// TIA Portal V16 export
// export: Created 2022-04-09T12:33:16.9078898Z, ExportSetting WithDefaults, DisplayName Totally Integrated Automation Portal, DisplayVersion V16 Update 3, DisplayName TIA Portal Version Control Interface, DisplayVersion V16 Update 2, DisplayName TIA Portal Openness, DisplayVersion V16 Update 3, DisplayName STEP 7 Professional, DisplayVersion V16 Update 3, DisplayName STEP 7 Safety, DisplayVersion V16, DisplayName WinCC Professional, DisplayVersion V16 Update 3
TYPE "UT22001_Dy_InstAnalogRead"
TITLE = Dynamic UDT [INSTRUMENTATION] — Analog Instrument Read, Scale and Monitor
// PRACTICAL SERIES AUTOMATION LIBRARY (PAL)   —   COPYRIGHT 2020 – M. GLEDHILL (MIT LICENCE)
//                   ———— ◆ ————
// FULL ONLINE DOCUMENTATION IS AVAILABLE AT: https://practicalseries.com/2001-pal/index.html
// stored: IsFailsafeCompliant false
   STRUCT
      revInfo : "UT01000_St_SysRevision";   // Revision information
      ___________0010_0 { ExternalAccessible := 'False'; ExternalVisible := 'False'; ExternalWritable := 'False'} : Int;
      ___________0010_1 { ExternalAccessible := 'False'; ExternalVisible := 'False'; ExternalWritable := 'False'} : Int;   // ▀▀▀▀ STATUS (FOR BLOCK ICON AND SYMBOL)
      status_ConfigError : Bool;   // STATUS — Block is configured incorrectly
      status_Alm_H : Bool;   // STATUS — High alarm is active (1 = alarm active, 0 = no alarm)
      status_Alm_L : Bool;   // STATUS — Low alarm is active (1 = alarm active, 0 = no alarm)
      status_Wrn_H : Bool;   // STATUS — High warning is active (1 = warning active, 0 = no warning)
      status_Wrn_L : Bool;   // STATUS — Low warning is active (1 = warning active, 0 = no warning)
      status_Alm_H_Mask : Bool;   // STATUS — High alarm is masked (1 = alarm masked, 0 = normal)
      status_Alm_L_Mask : Bool;   // STATUS — Low alarm is masked (1 = alarm masked, 0 = normal)
      status_Wrn_H_Mask : Bool;   // STATUS — High warning is masked (1 = warning masked, 0 = normal)
      status_Wrn_L_Mask : Bool;   // STATUS — Low warning is masked (1 = warning masked, 0 = normal)
      status_Alm_H_Dis : Bool;   // STATUS — High alarm is disabled (1 = alarm disabled, 0 = normal)
      status_Alm_L_Dis : Bool;   // STATUS — Low alarm is disabled (1 = alarm disabled, 0 = normal)
      status_Wrn_H_Dis : Bool;   // STATUS — High warning is disabled (1 = warning disabled, 0 = normal)
      status_Wrn_L_Dis : Bool;   // STATUS — Low warning is disabled (1 = warning disabled, 0 = normal)
      status_Fault : Bool;   // STATUS — Device is in fault (1 = fault present, 0 = healthy)
      status_SimOn : Bool;   // STATUS — Device is in simulation mode (1 = simulation mode on, 0 = normal)
      status_RemoteOn : Bool;   // STATUS — Device is in remote mode (1 = remote mode, 0 = remote mode off)
      status_LocalOn : Bool;   // STATUS — Device is in local mode (1 = local mode, 0 = local mode off)
      status_RLOff : Bool;   // STATUS — Remote/local mode disabled (1 = ALL mode on, 0 = RL mode selected)
      ___________0020_0 { ExternalAccessible := 'False'; ExternalVisible := 'False'; ExternalWritable := 'False'} : Int;
      ___________0020_1 { ExternalAccessible := 'False'; ExternalVisible := 'False'; ExternalWritable := 'False'} : Int;   // ▀▀▀▀ CALCULATED VALUES (ABSOLUTE OVER AND UNDER RANGE)
      cal_OR_Abs : Real;   // CALC — Over-range limit (absolute value)
      cal_UR_Abs : Real;   // CALC — Under-range limit (absolute value)
      ___________0030_0 { ExternalAccessible := 'False'; ExternalVisible := 'False'; ExternalWritable := 'False'} : Int;
      ___________0030_2 { ExternalAccessible := 'False'; ExternalVisible := 'False'; ExternalWritable := 'False'} : Int;   // ▀▀▀▀ OPERATING MODE SELECTION (FROM FACEPLATE OR PANEL)
      mode_Alm_H_MaskOn : Bool;   // MODE — Mask Alm_H (1 = mask alarm, 0 = normal)
      mode_Alm_L_MaskOn : Bool;   // MODE — Mask Alm_L (1 = mask alarm, 0 = normal)
      mode_Wrn_H_MaskOn : Bool;   // MODE — Mask Wrn_H (1 = mask warning, 0 = normal)
      mode_Wrn_L_MaskOn : Bool;   // MODE — Mask Wrn_H (1 = mask warning, 0 = normal)
      mode_SimOn : Bool := false;   // MODE — Simulation mode (1 = simulation mode active, 0 = normal)
      mode_SimValue : Real;   // MODE — Simulation value [engineering units]
      mode_RemoteOn : Bool := false;   // MODE — Local HMI control enabled (1 = control active, 0 = control disabled or N/A)
      mode_LocalOn : Bool := false;   // MODE — Remote SCADA control enabled (1 = control active, 0 = control disabled or N/A)
      ___________0040_0 { ExternalAccessible := 'False'; ExternalVisible := 'False'; ExternalWritable := 'False'} : Int;
      ___________0040_1 { ExternalAccessible := 'False'; ExternalVisible := 'False'; ExternalWritable := 'False'} : Int;   // ▀▀▀▀ MESSAGES (ALARMS, WARNINGS, FAULTS AND EVENTS)
      msg_Alm_H : Bool;   // MESSAGE — Alarm - high alarm is active
      msg_Alm_L : Bool;   // MESSAGE — Alarm - low alarm is active
      msg_Wrn_H : Bool;   // MESSAGE — Warning - high warning is active
      msg_Wrn_L : Bool;   // MESSAGE — Warning - low warning is active
      msg_Flt_External : Bool;   // MESSAGE — Fault - external fault signal is active
      msg_Flt_OverRange : Bool;   // MESSAGE — Fault - instrument is over-range
      msg_Flt_UnderRange : Bool;   // MESSAGE — Fault - instrument is under-range
      msg_Flt_OutOfRange : Bool;   // MESSAGE — Fault - instrument is out-of-range
      ___________0050_0 { ExternalAccessible := 'False'; ExternalVisible := 'False'; ExternalWritable := 'False'} : Int;
      ___________0050_1 { ExternalAccessible := 'False'; ExternalVisible := 'False'; ExternalWritable := 'False'} : Int;   // ▀▀▀▀ BATCH AND BOOKING DATA
      batch_ID : UInt;   // BATCH — Booking ID (optional for batch operations)
      ___________0060_0 { ExternalAccessible := 'False'; ExternalVisible := 'False'; ExternalWritable := 'False'} : Int;
      ___________0060_1 { ExternalAccessible := 'False'; ExternalVisible := 'False'; ExternalWritable := 'False'} : Int;   // ▀▀▀▀ LIVE DATA (SCALED READING & TIMER VALUES)
      actual_Value : Real;   // ACTUAL — SCALED INSTRUMENT VALUE [engineering units]
      actual_Alm_H_Timer : Real;   // ACTUAL — Timer value — alarm high operation timer [seconds]
      actual_Alm_L_Timer : Real;   // ACTUAL — Timer value — alarm low operation timer [seconds]
      actual_Wrn_H_Timer : Real;   // ACTUAL — Timer value — warning high operation timer [seconds]
      actual_Wrn_L_Timer : Real;   // ACTUAL — Timer value — warning low operation timer [seconds]
      ___________0090_0 { ExternalAccessible := 'False'; ExternalVisible := 'False'; ExternalWritable := 'False'} : Int;
      ___________0090_1 { ExternalAccessible := 'False'; ExternalVisible := 'False'; ExternalWritable := 'False'} : Int;   // ▀▀▀▀ BLOCK INTERNAL WORKING AND STORAGE AREA
      "$pret_AlmHEn" : Bool;   // INTERNAL — Edge retention (+ve) alarm high enable
      "$Pret_AlmLEn" : Bool;   // INTERNAL — Edge retention (+ve) alarm low enable
      "$pret_WrnHEn" : Bool;   // INTERNAL — Edge retention (+ve) warning high enable
      "$pret_WrnLEn" : Bool;   // INTERNAL — Edge retention (+ve) warning low enable
   END_STRUCT;
   // revInfo.REV_BLOCK := 'UT22001';
   // revInfo.REV_NUMBER := '001.102';
   // revInfo.REV_DATE := '2022-04-08';
   // revInfo.REV_AUTHOR := 'M. Gledhill';
END_TYPE
